Omron CX-Programmer project NewProject (CX-Programmer 9.61)

# PLC NewPLC1: CP1E N30

## Global symbols (name address type ; comment)
0.00 BOOL  ; TRIGGER W0 CONTACT
0.01 BOOL  ; PB 2 STOP
100.00 BOOL  ; PILOT LAMP
W0.00 BOOL  ; TRIGGER W0 CONTACT

## Program NewProgram1 (cyclic task 0)

### Section Section1

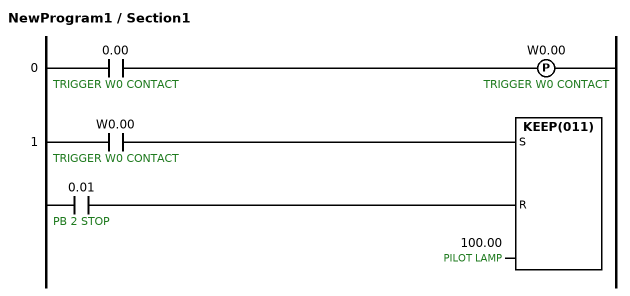
; rung 0
LD 0.00  ; TRIGGER W0 CONTACT
DIFU(013) W0.00  ; TRIGGER W0 CONTACT
; rung 1
LD W0.00  ; TRIGGER W0 CONTACT
LD 0.01  ; PB 2 STOP
KEEP(011) 100.00  ; PILOT LAMP

### Section END
; rung 0
END(001)